CASE actingLoadStep OF
	0:
		IF NOT actingStorage.findSlot(materialID := material, atSlot => slot) THEN //load from staging table
			fail := TRUE;
			RETURN;
		END_IF
		
		IF
			actingRobot.setCommandAndWait( //perform the task
				task:= A22.LOAD_CORNER_GUARD_LOWER,
				param1:= slot,
				param2:= 0,
				param3:= 0)
		THEN
			actingLoadStep := COMPLETE;
		END_IF
		
	COMPLETE:
		loadBottomLeft := TRUE;
END_CASE
END_METHOD

METHOD PROTECTED loadBottomRight : BOOL
VAR_IN_OUT
	actingRobot : Robot;
	actingStorage : MaterialStorage;
	actingLoadStep : INT;
END_VAR
VAR_INPUT
	material : STRING;
END_VAR
VAR_OUTPUT
	fail : BOOL;
END_VAR
VAR
	slot : INT;
END_VAR
IF material = '' THEN
	loadBottomRight := TRUE;
	RETURN;
END_IF

CASE actingLoadStep OF
	0:
		IF NOT actingStorage.findSlot(materialID := material, atSlot => slot) THEN //load from staging table
			fail := TRUE;
			RETURN;
		END_IF
		
		IF
			actingRobot.setCommandAndWait( //perform the task
				task:= A22.LOAD_CORNER_GUARD_LOWER,
				param1:= slot,
				param2:= 0,
				param3:= 0)
		THEN
			actingLoadStep := COMPLETE;
		END_IF
		
	COMPLETE:
		loadBottomRight := TRUE;
END_CASE
END_METHOD

METHOD PROTECTED loadCornerCardboards : BOOL
VAR_INPUT
	pair : REFERENCE TO PositionMaterials;
END_VAR
IF cornerSetLeft = 0 THEN //LEFT SIDE
	cornerSetLeft := Surface.TOP_RIGHT;
END_IF

IF
	leftRobotCornersSequence(
		actingRobot:= robotLeft, 
		skid:= skidLeft, 
		surfaceID:= cornerSetLeft,
		loadStep:= loadStepLeft, 
		materialID:= pair.topRight, 
		foldPos0:= currentBundle.cardboardFolds[cornerSetLeft][iPair],
		foldPos1:= 0,
		fail=> )
THEN
	CASE cornerSetLeft OF
		Surface.TOP_RIGHT: 
			cornerSetLeft := Surface.TOP_LEFT;
			loadStepLeft := 0;
			
		Surface.TOP_LEFT: 
			cornerSetLeft := Surface.BOTTOM_RIGHT;
			loadStepLeft := 0;
			
		Surface.BOTTOM_RIGHT: 
			cornerSetLeft := Surface.BOTTOM_LEFT;
			loadStepLeft := 0;
			
		Surface.BOTTOM_LEFT: 
			cornerSetLeft := COMPLETE;
			loadStepLeft := COMPLETE;
			
		COMPLETE:
			//
			
	END_CASE
END_IF



IF cornerSetRight = 0 THEN //RIGHT SIDE
	cornerSetRight := Surface.TOP_RIGHT;
END_IF

IF
	rightRobotCornersSequence(
		actingRobot:= robotRight, 
		skid:= skidRight, 
		loadStep:= loadStepRight, 
		materialID:= pair.topRight, 
		surfaceID:= cornerSetRight,
		foldPos1:= currentBundle.cardboardFolds[cornerSetRight][iPair], 
		foldPos2:= 0, 
		fail=> )
THEN
	CASE cornerSetRight OF
		Surface.TOP_RIGHT: 
			cornerSetRight := Surface.BOTTOM_RIGHT;
			loadStepRight := 0;
			
		Surface.BOTTOM_RIGHT: 
			cornerSetRight := COMPLETE;			
			loadStepRight := COMPLETE;
			
		COMPLETE:
			//
			
	END_CASE
END_IF


IF cornerSetLeft = COMPLETE AND cornerSetRight = COMPLETE THEN
	loadCornerCardboards := TRUE;
	
	loadStepLeft := loadStepRight := 0;
	cornerSetLeft := cornerSetRight := 0;
END_IF
END_METHOD

METHOD PROTECTED loadCornerGuards : BOOL
VAR_INPUT
	pair : REFERENCE TO PositionMaterials;
END_VAR
VAR_OUTPUT
	fail : BOOL;
END_VAR
VAR
	leftFail : BOOL;
	rightFail : BOOL;
END_VAR
CASE loadSet OF
	0: //upper corners
		IF 
			loadCornerGuardSequence(
				actingRobot:= robotLeft, 
				robotOutputs:= robotLeftOutputs, 
				actingStorage:= skidLeft, 
				actingLoadStep:= loadStepLeft, 
				surfaceID:= Surface.TOP_LEFT, 
				material:= pair.topLeft, 
				fail=> leftFail)
			AND
			loadCornerGuardSequence(
				actingRobot:= robotRight, 
				robotOutputs:= robotRightOutputs, 
				actingStorage:= skidRight,
				actingLoadStep:= loadStepRight, 
				surfaceID:= Surface.TOP_RIGHT, 
				material:= pair.topRight, 
				fail=> rightFail)
		THEN
			loadStepLeft := loadStepRight := 0;
			loadSet := 10;
		END_IF
		
	10: //lower corners
		IF 
			loadCornerGuardSequence(
				actingRobot:= robotLeft, 
				robotOutputs:= robotLeftOutputs, 
				actingStorage:= skidLeft, 
				actingLoadStep:= loadStepLeft, 
				surfaceID:= Surface.BOTTOM_LEFT, 
				material:= pair.bottomLeft, 
				fail=> leftFail)
			AND
			loadCornerGuardSequence(
				actingRobot:= robotRight, 
				robotOutputs:= robotRightOutputs, 
				actingStorage:= skidRight,
				actingLoadStep:= loadStepRight, 
				surfaceID:= Surface.BOTTOM_RIGHT, 
				material:= pair.bottomRight, 
				fail=> rightFail)
		THEN
			loadStepLeft := loadStepRight := 0;
			loadSet := COMPLETE;
		END_IF
	
	COMPLETE:
		loadStepLeft := loadStepRight := 0;
		loadSet := 0;
		
		loadCornerGuards := TRUE;
END_CASE

fail := MAX(leftFail, rightFail);
END_METHOD

METHOD loadCornerGuardSequence : BOOL
VAR_IN_OUT
	actingRobot : Robot;
	robotOutputs : ARRAY[1..50] OF INT;
	actingStorage : MaterialStorage;
	actingLoadStep : INT;
END_VAR
VAR_INPUT
	surfaceID : Surface;
	material : STRING;
END_VAR
VAR_OUTPUT
	fail : BOOL;
END_VAR
VAR
	slot : INT;
END_VAR
IF material = '' THEN
	loadCornerGuardSequence := TRUE;
	RETURN;
END_IF

CASE actingLoadStep OF
	0:
		IF NOT actingStorage.findSlot(materialID := material, atSlot => slot) THEN //load from staging table
			fail := TRUE;
			RETURN;
		END_IF
		
		MEMSET(ADR(robotOutputs), 0, SIZEOF(robotOutputs));
		CASE surfaceID OF
			Surface.TOP_LEFT, Surface.TOP_RIGHT: 		robotOutputs[1] := A22.LOAD_CORNER_GUARD_UPPER;
			Surface.BOTTOM_LEFT, Surface.BOTTOM_RIGHT:	robotOutputs[1] := A22.LOAD_CORNER_GUARD_LOWER;
		END_CASE
		robotOutputs[2] := slot;
		
		IF actingRobot.setParamsAndWait(robotOutputs) THEN
			actingLoadStep := COMPLETE;
		END_IF
		
	COMPLETE:
		//outerSuctions[surfaceID].enable := TRUE;
		loadCornerGuardSequence := TRUE;
END_CASE
END_METHOD

METHOD PROTECTED loadFlats : BOOL
VAR_INPUT
	pair : REFERENCE TO PositionMaterials;
END_VAR
CASE loadSet OF
	0: //top and bottom
		IF 
			loadTop(robotLeft, skidLeft, loadStepLeft, pair.top, fail=> ) AND
			loadBottom(robotRight, skidRight, loadStepRight, pair.bottom, fail=> )
		THEN
			loadStepLeft := loadStepRight := 0;
			loadSet := 10;
		END_IF
		
	10: //sides
		IF 
			loadSides(robotLeft, skidLeft, loadStepLeft, pair.top, fail=> ) AND
			loadSides(robotRight, skidRight, loadStepRight, pair.bottom, fail=> )
		THEN
			loadStepLeft := loadStepRight := 0;
			loadSet := COMPLETE;
		END_IF
	
	COMPLETE:
		loadStepLeft := loadStepRight := 0;
		loadSet := 0;
		
		loadFlats := TRUE;
END_CASE
END_METHOD

METHOD loadFlatSequence : BOOL
VAR_IN_OUT
	actingRobot : Robot;
	robotOutputs : ARRAY[1..50] OF INT;
	actingStorage : MaterialStorage;
	actingLoadStep : INT;
END_VAR
VAR_INPUT
	surfaceID : Surface;
	material : STRING;
END_VAR
VAR_OUTPUT
	fail : BOOL;
END_VAR
VAR
	slot : INT;
END_VAR
IF material = '' THEN
	loadFlatSequence := TRUE;
	RETURN;
END_IF

CASE actingLoadStep OF
	0:
		IF NOT actingStorage.findSlot(materialID := material, atSlot => slot) THEN
			fail := TRUE;
			RETURN;
		END_IF
		
		MEMSET(ADR(robotOutputs), 0, SIZEOF(robotOutputs));
		CASE surfaceID OF
			Surface.TOP: 					robotOutputs[1] := A22.LOAD_CARDBOARD_TOP;
			Surface.LEFT, Surface.RIGHT: 	robotOutputs[1] := A22.LOAD_CARDBOARD_SIDE;
			Surface.BOTTOM: 				robotOutputs[1] := A22.LOAD_CARDBOARD_BOTTOM;
		END_CASE
		robotOutputs[2] := slot;
		
		IF actingRobot.setParamsAndWait(robotOutputs) THEN
			actingLoadStep := COMPLETE;
		END_IF
		
	COMPLETE:
		loadFlatSequence := TRUE;
	
END_CASE
END_METHOD

METHOD PROTECTED loadSides : BOOL
VAR_IN_OUT
	actingRobot : Robot;
	actingStorage : MaterialStorage;
	actingLoadStep : INT;
END_VAR
VAR_INPUT
	material : STRING;
END_VAR
VAR_OUTPUT
	fail : BOOL;
END_VAR
VAR
	slot : INT;
END_VAR
IF material = '' THEN
	loadSides := TRUE;
	RETURN;
END_IF

CASE actingLoadStep OF
	0:
		IF NOT actingStorage.findSlot(materialID := material, atSlot => slot) THEN
			fail := TRUE;
			RETURN;
		END_IF
		
		IF
			actingRobot.setCommandAndWait( //perform the task
				task:= A22.LOAD_CARDBOARD_SIDE,
				param1:= slot,
				param2:= 0,
				param3:= 0)
		THEN
			actingLoadStep := COMPLETE;
		END_IF
		
	COMPLETE:
		//turn suction on
		loadSides := TRUE;
END_CASE
END_METHOD

METHOD PROTECTED loadTop : BOOL
VAR_IN_OUT
	actingRobot : Robot;
	actingStorage : MaterialStorage;
	actingLoadStep : INT;
END_VAR
VAR_INPUT
	material : STRING;
END_VAR
VAR_OUTPUT
	fail : BOOL;
END_VAR
VAR
	slot : INT;
END_VAR
IF material = '' THEN
	loadTop := TRUE;
	RETURN;
END_IF

CASE actingLoadStep OF
	0:
		IF NOT actingStorage.findSlot(materialID := material, atSlot => slot) THEN //load from staging table
			fail := TRUE;
			RETURN;
		END_IF
		
		IF
			actingRobot.setCommandAndWait( //perform the task
				task:= A22.LOAD_CARDBOARD_TOP,
				param1:= slot,
				param2:= 0,
				param3:= 0)
		THEN
			actingLoadStep := COMPLETE;
		END_IF
		
	COMPLETE:
		loadTop := TRUE;
END_CASE
END_METHOD

METHOD PROTECTED loadTopLeft : BOOL
VAR_IN_OUT
	actingRobot : Robot;
	actingStorage : MaterialStorage;
	actingLoadStep : INT;
END_VAR
VAR_INPUT
	material : STRING;
END_VAR
VAR_OUTPUT
	fail : BOOL;
END_VAR
VAR
	slot : INT;
END_VAR
IF material = '' THEN
	loadTopLeft := TRUE;
	RETURN;
END_IF

CASE actingLoadStep OF
	0:
		IF NOT actingStorage.findSlot(materialID := material, atSlot => slot) THEN //load from staging table
			fail := TRUE;
			RETURN;
		END_IF
		
		IF
			actingRobot.setCommandAndWait( //perform the task
				task:= A22.LOAD_CORNER_GUARD_UPPER,
				param1:= slot,
				param2:= 0,
				param3:= 0)
		THEN
			actingLoadStep := COMPLETE;
		END_IF
		
	COMPLETE:
		loadTopLeft := TRUE;
END_CASE
END_METHOD

METHOD PROTECTED loadTopRight : BOOL
VAR_IN_OUT
	actingRobot : Robot;
	actingStorage : MaterialStorage;
	actingLoadStep : INT;
END_VAR
VAR_INPUT
	material : STRING;
END_VAR
VAR_OUTPUT
	fail : BOOL;
END_VAR
VAR
	slot : INT;
END_VAR
IF material = '' THEN
	loadTopRight := TRUE;
	RETURN;
END_IF

CASE actingLoadStep OF
	0:
		IF NOT actingStorage.findSlot(materialID := material, atSlot => slot) THEN //load from staging table
			fail := TRUE;
			RETURN;
		END_IF
		
		IF
			actingRobot.setCommandAndWait( //perform the task
				task:= A22.LOAD_CORNER_GUARD_UPPER,
				param1:= slot,
				param2:= 0,
				param3:= 0)
		THEN
			actingLoadStep := COMPLETE;
		END_IF
		
	COMPLETE:
		loadTopRight := TRUE;
END_CASE
END_METHOD

METHOD placeFrontCover : BOOL
VAR_INPUT
END_VAR
END_METHOD

METHOD PROTECTED process : BOOL
VAR
	masterLength : REAL;
	targetPos : REAL;
	targetStep : INT;
END_VAR
VAR
	maxHeight : REAL := 1000; //1000mm, 100cm, 1m tall at home pos
END_VAR
(*
VAR_INST
	resumePosition : REAL;
END_VAR
VAR CONSTANT
	wrapDelta : REAL := 5;
END_VAR
*)
//TODO: write instructions for wrapping front and back covers

IF NOT frontCoverPlaced THEN
	targetPos := 0;
	
ELSIF iPair < GVL.maxPairs THEN
	targetPos := currentPair.position;
	
ELSIF NOT backCoverPlaced AND iPair >= GVL.maxPairs THEN
	targetPos := currentBundle.length;
	
ELSIF iPair >= GVL.maxPairs THEN
	process := TRUE;
	RETURN;
	
END_IF

CASE step OF
	PLACE_FRONT_COVER:
		IF placeFrontCover() THEN
			step := RUN_TO_POSITION;
		END_IF
	
	RUN_TO_POSITION:
		IF //only load corners, flats will be PUSHed when bundle arrives at position
			directionCheckAndSet(pushConveyorPos, currentPair.position) AND 
			load(pair:= currentPair)
		THEN
			step := 10;
		END_IF
		
	LOAD_FLATS:
		IF loadFlats(pair:= currentPair) THEN
			step := PUSH;
		END_IF
		
	PUSH:
		setConveyorMode(ConveyorMode.STOP);
		(*
		IF
			NOT insertionLeft.align(targetPos:= maxHeight - currentBundle.height) OR
			NOT insertionRight.align(targetPos:= maxHeight - currentBundle.height)
		THEN
			RETURN;
		END_IF
		
		insertionLeft.press();
		insertionRight.press();
		*)
		
		IF NOT insertionLeft.contact THEN
			//insertionRight.slideOut();
			insertionLeft.traverse(direction:= MC_Negative_Direction);
			insertionLeft.press();
		END_IF
		
		IF NOT insertionRight.contact THEN
			//insertionRight.slideOut();
			insertionRight.traverse(direction:= MC_Negative_Direction);
			insertionRight.press();
		END_IF
		
		(*
		IF NOT insertionBottom.contact THEN
			insertionBottom.traverse(direction := FALSE);
		END_IF
		*)
		
		IF insertionLeft.contact AND insertionRight.contact (*AND insertionBottom.contact*) THEN		
			step := RUN_TO_WRAP_POSITION;
		END_IF
		
	RUN_TO_WRAP_POSITION:
		masterLength := GetPositionMasterLength(currentPair);
		IF iWrap >= currentPair.wrapPoints THEN
			step := COMPLETE;
			RETURN;
		END_IF
		
		IF //compare current position with wrap position
			directionCheckAndSet(
				wrapConveyorPos,
				(currentPair.position - masterLength/2) + (masterLength/(currentPair.wrapPoints + 1) * (iWrap + 1)))
		THEN
			step := WRAP_AND_RELEASE;
		END_IF
		
	WRAP_AND_RELEASE: //wrap
		setConveyorMode(ConveyorMode.STOP);
		IF wrapper.ready OR (NOT wrapper.busy AND NOT wrapper.error) THEN
			wrapper.wrap(currentPair.wrapRotations);
		END_IF
		
		IF NOT insertionLeft.home THEN
			insertionLeft.align(0);
			insertionLeft.release();
		END_IF
		
		IF NOT insertionRight.home THEN
			insertionRight.align(0);
			insertionRight.release();
		END_IF
		
		IF wrapper.done AND insertionLeft.home AND insertionRight.home (*AND insertionBottom.home*) THEN
			step := WRAP_AND_RELEASE;
		END_IF
		
	COMPLETE: //reset
		setConveyorMode(ConveyorMode.FORWARD);
		
		iPair := iPair + 1;
		IF iPair >= GVL.maxPairs THEN
			iPair := 0;
			process := TRUE;
		END_IF
		iWrap := 0;
		
		step := 0;
END_CASE
END_METHOD

METHOD PROTECTED rightRobotCornersSequence : BOOL
VAR_IN_OUT
	actingRobot : Robot;
	skid : MaterialStorage;
	loadStep : INT;
END_VAR
VAR_INPUT
	surfaceID : Surface;
	materialID : STRING;
	foldPos1 : INT;
	foldPos2 : INT;
END_VAR
VAR_OUTPUT
	fail : BOOL;
END_VAR
VAR
	slot : INT;
	
	task : INT;
	param0, param1, param2 : INT;
END_VAR
IF materialID = '' THEN
	rightRobotCornersSequence := TRUE;
	RETURN;
END_IF

CASE loadStep OF
	0: //overhead to insertion
		IF overhead = '' THEN
			RETURN;
		END_IF
		
		CASE surfaceID OF
			Surface.TOP_RIGHT:
				task := A22.LOAD_OVERHEAD_TO_UPPER_CORNER;
				
			Surface.BOTTOM_RIGHT:
				task := A22.LOAD_OVERHEAD_TO_LOWER_CORNER;
				
		END_CASE
		
		IF
			actingRobot.setCommandAndWait(
				task:= task, 
				param1:= slot, 
				param2:= foldPos1, 
				param3:= foldPos2)
		THEN
			loadStep := COMPLETE;
		END_IF
	
	COMPLETE:
		//turn on suction
		rightRobotCornersSequence := TRUE;
	
END_CASE
END_METHOD

METHOD PROTECTED robotsFailed : BOOL
VAR_INPUT
END_VAR
IF NOT robotLeft.operational OR NOT robotLeft.operational THEN
	error := TRUE;
	currentBypass := TRUE;
	robotsFailed := TRUE;
END_IF
END_METHOD

METHOD PROTECTED setOrder : BOOL
VAR_IN_OUT
	innerArray : ARRAY[*] OF PositionMaterials;
	outerArray : ARRAY[*] OF PositionMaterials;
	
	combined : ARRAY[*] OF PositionMaterials;
	
	i_inner : INT;
	i_outer : INT;
	i_combined : INT;
END_VAR
VAR
	topLength : REAL;
	leftLength : REAL;
	rightLength : REAL;
	bottomLength : REAL;
	
	topLeftLength : REAL;
	topRightLength : REAL;
	bottomLeftLength : REAL;
	bottomRightLength : REAL;
	
	outerMaterialLength : REAL;
	innerMaterialLength : REAL;
END_VAR
//if inner material is in front of outer material, inner material goes first
IF innerArray[i_inner].position <= outerArray[i_outer].position THEN

	combined[i_combined] := innerArray[i_inner];
	i_inner := i_inner + 1; //check next cardboard during next iteration
	
	setOrder := TRUE;
	RETURN;
END_IF
	
outerMaterialLength := GetPositionMasterLength(outerArray[i_outer]);
innerMaterialLength := GetPositionMasterLength(innerArray[i_inner]);

//if current inner material is too close to current outer material, place inner material first
//compare inner materials' front with outer material's back
IF (innerArray[i_inner].position - innerMaterialLength/2) < (outerArray[i_outer].position + outerMaterialLength/2) THEN
	combined[i_combined] := innerArray[i_inner];
	i_inner := i_inner + 1;
ELSE //otherwise, outer material can go
	combined[i_combined] := outerArray[i_outer];
	i_outer := i_outer + 1;
END_IF

setOrder := TRUE;
END_METHOD

METHOD PROTECTED usesProcess : BOOL
VAR
	i : INT;
END_VAR
IF materialsArr = 0 THEN
	RETURN;
END_IF

FOR i:=0 TO GVL.maxPairs BY 1 DO
	IF PositionIsValid(materialsArr[i]) THEN
		usesProcess := TRUE;
		RETURN;		
	END_IF
END_FOR
END_METHOD

END_FUNCTION_BLOCK

// ---- Sections/Concrete/ChipboardEx.TcPOU
FUNCTION_BLOCK ChipboardEx EXTENDS SectionEx
VAR
	robotLeft, robotRight : REFERENCE TO Robot;
	
	skidLeft, skidRight : REFERENCE TO MaterialStorage;
	
	toolStorageLeft, toolStorageRight : REFERENCE TO A21ToolStorage;
END_VAR
VAR
	pushSmallConveyorPos : REAL;
	pushLargeConveyorPos : REAL;
	
	topCIP : STRING;
	bottomCIP : STRING;
	
	materialsArr : POINTER TO PositionMaterials; //array of PositionMaterials
	//currentPair : REFERENCE TO PositionMaterials;	
	
	step : (RUN_TO_POSITION, LOAD_MATERIAL, PUSH, RESET);
	
	robotLeftOutputs, robotRightOutputs : ARRAY[1..50] OF INT;
END_VAR

entryRefPos := pushSmallConveyorPos;
exitRefPos := pushLargeConveyorPos;

SUPER^();

CASE status OF
	SectionStatus.IDLE:
		//RETURN;
	
	SectionStatus.ALIGNING:
		//
		
	SectionStatus.ACTIVE:
		//
		
	SectionStatus.CLEARING:
		//
		
	SectionStatus.COMPLETE:	
		//
		
	-100:
		RETURN;
		
END_CASE
	
materialsArr := ADR(currentBundle.chipboard);

loaded := 
	topCIP = materialsArr[iPair].top AND
	bottomCIP = materialsArr[iPair].bottom;
	
IF NOT(robotLeft.operational AND robotRight.operational) THEN
	currentBypass := TRUE;
END_IF

METHOD changeRobotsEOAT : BOOL
VAR_INPUT
END_VAR
IF robotLeft.tool <> sectionID THEN
	MEMSET(ADR(robotLeftOutputs), 0, SIZEOF(robotLeftOutputs));
	robotLeftOutputs[1] := A21.TOOL_CHANGE_CHIPBOARD;
	robotLeft.setParamsAndWait(robotLeftOutputs);
END_IF

IF robotRight.tool <> sectionID THEN
	MEMSET(ADR(robotRightOutputs), 0, SIZEOF(robotRightOutputs));
	robotRightOutputs[1] := A21.TOOL_CHANGE_CHIPBOARD;
	robotRight.setParamsAndWait(robotRightOutputs);
END_IF

changeRobotsEOAT := robotLeft.tool = sectionID AND robotRight.tool = sectionID;
END_METHOD

METHOD initHardware : BOOL
conveyors := ADR(allConveyors);

robotLeft REF= robots[1];
robotRight REF= robots[2];

skidLeft REF= chipboardSkidLeft;
skidRight REF= chipboardSkidRight;
END_METHOD

METHOD PROTECTED load : BOOL
VAR_INPUT
	pair : REFERENCE TO PositionMaterials;
END_VAR
(*
top:
	grab chipboard
	move chipboard to top

bottom:
	grab chipboard and lower conveyor
	move chipboard to lowered conveyor
	which conveyor depends on size of chipboard
	raise conveyor
*)
IF NOT (robotLeft.reserve(sectionID) AND robotRight.reserve(sectionID)) THEN
	RETURN;
END_IF

IF NOT (robotLeft.tool = sectionID AND robotRight.tool = sectionID) THEN //robots have wrong tool
	changeRobotsEOAT(); //wait for robots to finish changing tools
	RETURN;
END_IF
//continues once both robots have correct tool

CASE loadSet OF
	0: //top and bottom
		IF 
			loadingSequence(
				actingRobot:= robotLeft, 
				robotOutputs:= robotLeftOutputs, 
				storage:= skidLeft, 
				loadStep:= loadStepLeft, 
				surfaceID:= Surface.TOP,
				material:= pair.top, 
				fail=> )
			AND
			loadingSequence(
				actingRobot:= robotRight, 
				robotOutputs:= robotRightOutputs, 
				storage:= skidRight, 
				loadStep:= loadStepRight, 
				surfaceID:= Surface.TOP,
				material:= pair.bottom, 
				fail=> )
		THEN
			loadStepLeft := loadStepRight := 0;
			loadSet := 10;
		END_IF
		
	10 : //recovery
		IF robotLeft.operational AND NOT robotRight.operational THEN //left ok, right fail
			IF
				loadingSequence(
					actingRobot:= robotLeft, 
					robotOutputs:= robotLeftOutputs, 
					storage:= skidLeft, 
					loadStep:= loadStepLeft, 
					surfaceID:= Surface.BOTTOM,
					material:= pair.top, 
					fail=> ) //load bottom with left robot
			THEN
				step := COMPLETE;
			END_IF
			
		ELSIF NOT robotLeft.operational AND robotRight.operational THEN //left fail, right ok
			IF
				loadingSequence(
					actingRobot:= robotRight, 
					robotOutputs:= robotRightOutputs, 
					storage:= skidRight, 
					loadStep:= loadStepRight, 
					surfaceID:= Surface.TOP,
					material:= pair.bottom, 
					fail=> ) //load top with right robot
			THEN
				step := COMPLETE;
			END_IF
			
		ELSE
			error := TRUE;
			currentBypass := TRUE;
				
		END_IF
		
		loadSet := COMPLETE;
		
	COMPLETE:
		loadSet := 0;
		
		loaded := 
			topCip = pair.top AND
			bottomCip = pair.bottom;
			
		robotLeft.release(sectionID);
		robotRight.release(sectionID);
			
		load := TRUE;
END_CASE
END_METHOD

METHOD loadBottom : BOOL
VAR_IN_OUT
	actingRobot : Robot;
	robotReserved : BOOL;
	robotOutputs : ARRAY[1..50] OF INT;
	actingStorage : MaterialStorage;
	actingLoadStep : INT;
END_VAR
VAR_INPUT
	material : STRING;
END_VAR
VAR_OUTPUT
	fail : BOOL;
END_VAR
VAR
	done : BOOL;
END_VAR
VAR
	slot : INT;
END_VAR
IF material = '' THEN
	step := COMPLETE;
END_IF

IF actingLoadStep <> COMPLETE AND_THEN NOT actingRobot.reserve(sectionID) THEN
	RETURN;
END_IF

CASE actingLoadStep OF
	0:
		IF NOT actingStorage.findSlot(materialID := material, atSlot => slot) THEN
			fail := TRUE;
			RETURN;
		END_IF
		
		MEMSET(ADR(robotOutputs), 0, SIZEOF(robotOutputs));
		robotOutputs[1] := A21.GET_CHIPBOARD_FROM_SKID;
		robotOutputs[2] := slot;
		
		IF actingRobot.setParamsAndWait(robotOutputs) THEN
			actingLoadStep := 10;
		END_IF
		
	10:
		MEMSET(ADR(robotOutputs), 0, SIZEOF(robotOutputs));
		robotOutputs[1] := A21.PLACE_CHIPBOARD_TO_BOTTOM;
		robotOutputs[2] := slot;
		
		IF actingRobot.setParamsAndWait(robotOutputs) THEN
			actingLoadStep := 10;
		END_IF
		
	COMPLETE:
		actingRobot.release(sectionID);
		loadBottom := TRUE;
		
END_CASE
END_METHOD

METHOD loadingSequence : BOOL
VAR_IN_OUT
	actingRobot : Robot;
	robotOutputs : ARRAY[1..50] OF INT;
	storage : MaterialStorage;
	loadStep : INT;
END_VAR
VAR_INPUT
	surfaceID : Surface;
	material : STRING;
END_VAR
VAR_OUTPUT
	fail : BOOL;
END_VAR
VAR
	slot : INT;
END_VAR
IF material = '' THEN
	loadingSequence := TRUE;
	RETURN;
END_IF

CASE loadStep OF
	0:
		IF NOT storage.findSlot(materialID := material, atSlot => slot) THEN
			fail := TRUE;
			RETURN;
		END_IF
		
		MEMSET(ADR(robotOutputs), 0, SIZEOF(robotOutputs));
		robotOutputs[1] := A21.GET_CHIPBOARD_FROM_SKID;
		robotOutputs[2] := slot;
		
		CASE surfaceID OF
			Surface.TOP:
				IF actingRobot.setParamsAndWait(robotOutputs) THEN
					loadStep := 10;
				END_IF
				
			Surface.BOTTOM:
				//lower conveyor
				IF actingRobot.setParamsAndWait(robotOutputs) (*AND conveyor lowered*) THEN
					loadStep := 10;
				END_IF
			
		END_CASE
		
	10:
		MEMSET(ADR(robotOutputs), 0, SIZEOF(robotOutputs));
		CASE surfaceID OF
			Surface.TOP: 					robotOutputs[1] := A21.PLACE_CHIPBOARD_TO_TOP;
			Surface.BOTTOM: 				robotOutputs[1] := A21.PLACE_CHIPBOARD_TO_BOTTOM;
		END_CASE
		robotOutputs[2] := slot;
		
		IF actingRobot.setParamsAndWait(robotOutputs) THEN
			loadStep := 10;
		END_IF
		
	COMPLETE:
		actingRobot.release(sectionID);
		loadingSequence := TRUE;
		
END_CASE
END_METHOD

METHOD loadTop : BOOL
VAR_IN_OUT
	actingRobot : Robot;
	robotOutputs : ARRAY[1..50] OF INT;
	actingStorage : MaterialStorage;
	actingLoadStep : INT;
END_VAR
VAR_INPUT
	material : STRING;
END_VAR
VAR_OUTPUT
	fail : BOOL;
END_VAR
VAR
	slot : INT;
END_VAR
IF actingLoadStep <> COMPLETE AND_THEN NOT actingRobot.reserve(sectionID) THEN
	RETURN;
END_IF

CASE actingLoadStep OF
	0: //grab chipboard
		IF NOT actingStorage.findSlot(materialID := material, atSlot => slot) THEN
			fail := TRUE;
			RETURN;
		END_IF
		
		MEMSET(ADR(robotOutputs), 0, SIZEOF(robotOutputs));
		robotOutputs[1] := A21.GET_CHIPBOARD_FROM_SKID;
		robotOutputs[2] := slot;
		
		IF actingRobot.setParamsAndWait(robotOutputs) THEN
			actingLoadStep := 10;
		END_IF
		
	10: //load chipboard
		MEMSET(ADR(robotOutputs), 0, SIZEOF(robotOutputs));
		robotOutputs[1] := A21.PLACE_CHIPBOARD_TO_TOP;
		robotOutputs[2] := slot;
		
		IF actingRobot.setParamsAndWait(robotOutputs) THEN
			actingLoadStep := 10;
		END_IF
		
	COMPLETE:
		actingRobot.release(sectionID);
		loadTop := TRUE;
		
END_CASE
END_METHOD

METHOD PROTECTED process : BOOL
VAR
	currentPair : REFERENCE TO PositionMaterials REF= materialsArr[iPair];
END_VAR
VAR_INST
	cmdSent : BOOL;
	
	test : BOOL;
	
	i : INT;
	conveyorsExtended : BOOL := TRUE;
END_VAR
IF iPair >= GVL.maxPairs THEN
	process := TRUE;
	RETURN;
END_IF

CASE step OF
	RUN_TO_POSITION: //free run until position reached
		IF directionCheckAndSet(pushSmallConveyorPos, currentPair.position) THEN
			step := PUSH;
		END_IF
		
	LOAD_MATERIAL: //loading must be done when bundle reaches position, not before
		setConveyorMode(ConveyorMode.STOP); //request stop at position
		IF load(currentPair) THEN
			step := PUSH;
		END_IF
	
	PUSH: //push materials
		setConveyorMode(ConveyorMode.STOP); //request stop at position
		FOR i:=firstConveyor TO lastConveyor BY 1 DO
			IF NOT conveyors[i].extended THEN
				conveyors[i].extend();
			END_IF
			conveyorsExtended := MIN(conveyorsExtended, conveyors[i].extended);
		END_FOR
		
		IF conveyorsExtended THEN
			step := RESET;
		END_IF
		
	RESET: //finished at this position, reset
		setConveyorMode(ConveyorMode.FORWARD);
		cmdSent := FALSE;
		
		iPair := iPair + 1;
		
		step := 0;
END_CASE
END_METHOD

METHOD PROTECTED usesProcess : BOOL
VAR
	i : INT;
END_VAR
IF materialsArr = 0 THEN
	RETURN;
END_IF

FOR i:=0 TO GVL.maxPairs BY 1 DO
	IF PositionIsValid(materialsArr[i]) THEN
		usesProcess := TRUE;
		RETURN;		
	END_IF
END_FOR
END_METHOD

END_FUNCTION_BLOCK

// ---- Sections/Concrete/WoodBunkEx.TcPOU
FUNCTION_BLOCK WoodBunkEx EXTENDS SectionEx
VAR //references to objects imported from Hardware GVL - using references instead of VAR_EXTERNAL or direct access allows local renaming
	robotLeft, robotRight : REFERENCE TO Robot;
	
	stagingTableLeft, stagingTableRight : REFERENCE TO WoodBunkTable;
	magazineLeft, magazineRight: REFERENCE TO MaterialStorage;
	
	strapper : REFERENCE TO StrapMachine;
	
	insertionLeft, insertionRight : REFERENCE TO Insertion;
	insertionBottom : REFERENCE TO AirPiston;
	
	toolStorageLeft, toolStorageRight : REFERENCE TO A21ToolStorage;
END_VAR
VAR
	conveyorPos : REAL;
	
	insertionSlots : ARRAY[Surface.TOP..Surface.BOTTOM] OF STRING;
	
	materialsArr : POINTER TO PositionMaterials; //array of PositionMaterials
	currentPair : REFERENCE TO PositionMaterials;
	
	stagingMaterial : STRING; //ex: currentPair.left
	currentMaterial : STRING; //ex: WDS18_WDS20 --> WDS18, then WDS20
	
	stagingTemplateReady : BOOL;
	stagingTemplateLeft : WoodBunkTable;
	stagingTemplateRight : WoodBunkTable;
	
	step : (RUN_TO_POSITION, PUSH, RUN_TO_STRAP, STRAP, RELEASE, RESET);
	
	//for staging use
	stageSet : INT;	
	stageStepLeft, stageStepRight : INT;
	iStagingSlotLeft, iStagingSlotRight : INT;
	
	robotLeftOutputs, robotRightOutputs : ARRAY[1..50] OF INT;
END_VAR
VAR
	tempInspectionSuite : VisionSuite; //send/receive from TcpServer
	leftInspectionFrame, rightInspectionFrame : VisionFrame; //parsed from above
END_VAR
VAR CONSTANT
	leftCamera : INT := 1;
	rightCamera : INT := 2;
END_VAR

entryRefPos := conveyorPos;
exitRefPos := conveyorPos;

SUPER^();

CASE status OF
	SectionStatus.IDLE:
		//RETURN;
	
	SectionStatus.ALIGNING:
		//
		
	SectionStatus.ACTIVE:
		//
		
	SectionStatus.CLEARING:
		stagingTemplateReady := FALSE;
		
	SectionStatus.COMPLETE:	
		//
		
	-100:
		RETURN;
		
END_CASE

materialsArr := ADR(currentBundle.woodBunk);

loaded := 
	insertionSlots[Surface.TOP] = materialsArr[iPair].top AND
	insertionSlots[Surface.LEFT] = materialsArr[iPair].left AND
	insertionSlots[Surface.RIGHT] = materialsArr[iPair].right AND
	insertionSlots[Surface.BOTTOM] = materialsArr[iPair].bottom;
	
//bundle needs this section's materials, and either robot failed
IF usesProcess() AND NOT(robotLeft.operational AND robotRight.operational) THEN 

	currentBypass := TRUE;
	RETURN;
END_IF //otherwise, carry over bypass from prev section

stage();

METHOD changeRobotsEOAT : BOOL
VAR_INPUT
END_VAR
IF robotLeft.tool <> sectionID THEN
	MEMSET(ADR(robotLeftOutputs), 0, SIZEOF(robotLeftOutputs));
	robotLeftOutputs[1] := A21.TOOL_CHANGE_CHIPBOARD;
	robotLeft.setParamsAndWait(robotLeftOutputs);
END_IF

IF robotRight.tool <> sectionID THEN
	MEMSET(ADR(robotRightOutputs), 0, SIZEOF(robotRightOutputs));
	robotRightOutputs[1] := A21.TOOL_CHANGE_CHIPBOARD;
	robotRight.setParamsAndWait(robotRightOutputs);
END_IF

changeRobotsEOAT := robotLeft.tool = sectionID AND robotRight.tool = sectionID;
END_METHOD

METHOD PROTECTED createStagingTemplate : BOOL
VAR
	remainingMaterial : STRING;
	splitMaterial : STRING;
	
	i : INT;
END_VAR
FOR i:=0 TO GVL.maxPairs BY 1 DO //iterate through all pairs and autofill the template
	//LEFT TABLE
	remainingMaterial := materialsArr[i].top;
	WHILE FIND(remainingMaterial, '_') > 0 DO //until no underscore found
		splitCombinedMaterials(remainingMaterial, splitMaterial);
		stagingTemplateLeft.autofill(splitMaterial);
	END_WHILE
	stagingTemplateLeft.autofill(remainingMaterial);
	
	remainingMaterial := materialsArr[i].left;
	WHILE FIND(remainingMaterial, '_') > 0 DO
		splitCombinedMaterials(remainingMaterial, splitMaterial);
		stagingTemplateLeft.autofill(splitMaterial);
	END_WHILE
	stagingTemplateLeft.autofill(remainingMaterial);
	
	//RIGHT TABLE
	remainingMaterial := materialsArr[i].right;
	WHILE FIND(remainingMaterial, '_') > 0 DO
		splitCombinedMaterials(remainingMaterial, splitMaterial);
		stagingTemplateRight.autofill(splitMaterial);
	END_WHILE
	stagingTemplateRight.autofill(remainingMaterial);
	
	remainingMaterial := materialsArr[i].bottom;
	WHILE FIND(remainingMaterial, '_') > 0 DO
		splitCombinedMaterials(remainingMaterial, splitMaterial);
		stagingTemplateRight.autofill(splitMaterial);
	END_WHILE
	stagingTemplateRight.autofill(remainingMaterial);
END_FOR
END_METHOD

METHOD findOpenSlot : BOOL
VAR_INPUT
	materialCode : STRING;
END_VAR
VAR_OUTPUT
	openSlot : INT := 0;
END_VAR
(*
IF FIND(materialCode, 'WDW') > 0 THEN //top wide, load in slot 0-1
	FOR i:=1 TO 2 BY 1 DO
		IF stageTableLeft[i] = '' THEN
			findOpenSlot := TRUE;
			openSlot := i;
			RETURN;
		END_IF
	END_FOR
	
ELSIF FIND(materialCode, 'WDT') > 0 OR FIND(materialCode, 'WDS') > 0 THEN //top std and sides, load in slot 2-9
	FOR i:=3 TO 10 BY 1 DO
		IF stageTableLeft[i] = '' THEN
			findOpenSlot := TRUE;
			openSlot := i;
			RETURN;
		END_IF
	END_FOR
	
END_IF
*)
END_METHOD

METHOD initHardware : BOOL
conveyors := ADR(allConveyors);

robotLeft REF= robots[1];
robotRight REF= robots[2];

strapper REF= strapperA21;

insertionLeft REF= insertionA21Left;
insertionLeft REF= insertionA21Right;

stagingTableLeft REF= stagingTableLeft;
stagingTableRight REF= stagingTableRight;

magazineLeft REF= woodBunkMagazineLeft;
magazineRight REF= woodBunkMagazineRight;

(*
strapper REF= Hardware.strapper;

insertionLeft REF= Hardware.insertionWoodBunkSides[Surface.LEFT];
insertionLeft REF= Hardware.insertionWoodBunkSides[Surface.RIGHT];

stagingTableLeft REF= Hardware.stagingTable[Surface.LEFT];
stagingTableRight REF= Hardware.stagingTable[Surface.RIGHT];

magazineLeft REF= Hardware.woodBunkMagazine[Surface.LEFT];
magazineRight REF= Hardware.woodBunkMagazine[Surface.RIGHT];
*)
END_METHOD

METHOD PROTECTED load : BOOL
VAR_INPUT
	pair : REFERENCE TO PositionMaterials;
END_VAR
IF NOT robotLeft.operational OR NOT robotLeft.operational THEN
	error := TRUE;
	
	currentBypass := TRUE;
	RETURN;
END_IF

IF NOT (robotLeft.reserve(sectionID) AND robotRight.reserve(sectionID)) THEN
	RETURN;
END_IF

IF NOT (robotLeft.tool = sectionID AND robotRight.tool = sectionID) THEN //robots have wrong tool
	changeRobotsEOAT(); //wait for robots to finish changing tools
	RETURN;
END_IF


CASE loadSet OF
	0: //top and bottom
		IF 
			loadingSequence(
				actingRobot:= robotLeft, 
				robotOutputs:= robotLeftOutputs, 
				stagingTable:= stagingTableLeft, 
				loadStep:= loadStepLeft, 
				surfaceID:= Surface.TOP, 
				material:= pair.top, 
				fail=> )
			AND
			loadingSequence(
				actingRobot:= robotRight, 
				robotOutputs:= robotRightOutputs, 
				stagingTable:= stagingTableRight, 
				loadStep:= loadStepRight, 
				surfaceID:= Surface.BOTTOM, 
				material:= pair.bottom, 
				fail=> )
		THEN
			loadStepLeft := loadStepRight := 0;
			loadSet := 10;
		END_IF
		
	10: //sides
		IF
			loadingSequence(
				actingRobot:= robotLeft, 
				robotOutputs:= robotLeftOutputs, 
				stagingTable:= stagingTableLeft, 
				loadStep:= loadStepLeft, 
				surfaceID:= Surface.LEFT, 
				material:= pair.left, 
				fail=> )
			AND
			loadingSequence(
				actingRobot:= robotRight, 
				robotOutputs:= robotRightOutputs, 
				stagingTable:= stagingTableRight, 
				loadStep:= loadStepRight, 
				surfaceID:= Surface.RIGHT, 
				material:= pair.right, 
				fail=> )
		THEN
			loadStepLeft := loadStepRight := 0;
			loadSet := COMPLETE;
		END_IF
		
	COMPLETE:
		loadSet := 0;
		loadStepLeft := loadStepRight := 0;
		
		loaded := 
			insertionSlots[Surface.TOP] = materialsArr[iPair].top AND
			insertionSlots[Surface.LEFT] = materialsArr[iPair].left AND
			insertionSlots[Surface.RIGHT] = materialsArr[iPair].right AND
			insertionSlots[Surface.BOTTOM] = materialsArr[iPair].bottom;
		
		robotLeft.release(sectionID);
		robotRight.release(sectionID);
		
		load := TRUE;
END_CASE
END_METHOD

METHOD loadBottom : BOOL
VAR_IN_OUT //acting refers to which robot is performing the task, if the designated robot fails the other may take over
	actingRobot : Robot;
	robotOutputs : ARRAY[1..50] OF INT;
	actingStagingTable : WoodBunkTable;
	actingLoadStep : INT;
END_VAR
VAR_INPUT
	material : STRING;
END_VAR
VAR_OUTPUT
	fail : BOOL;
END_VAR
VAR
	slot : INT;
END_VAR
IF
	actingLoadStep <> COMPLETE AND_THEN
	NOT actingRobot.reserve(sectionID)
THEN
	RETURN;
END_IF

CASE actingLoadStep OF
	0:
		IF NOT actingStagingTable.findSlot(materialID := material, atSlot => slot) THEN
			fail := TRUE;
			RETURN;
		END_IF
		
		MEMSET(ADR(robotOutputs), 0, SIZEOF(robotOutputs));
		robotOutputs[1] := A21.LOAD_BUNK_TO_BOTTOM;
		robotOutputs[2] := slot;
		
		IF actingRobot.setParamsAndWait(robotOutputs) THEN
			actingLoadStep := COMPLETE;
		END_IF
		
	COMPLETE:
		//turn suction on
		actingRobot.release(sectionID);
		loadBottom := TRUE;
END_CASE
END_METHOD

METHOD loadingSequence : BOOL
VAR_IN_OUT
	actingRobot : Robot;
	robotOutputs : ARRAY[1..50] OF INT;
	stagingTable : WoodBunkTable;
	loadStep : INT;
END_VAR
VAR_INPUT
	surfaceID : Surface;
	material : STRING;
END_VAR
VAR_OUTPUT
	fail : BOOL;
END_VAR
VAR
	slot : INT;
END_VAR
IF material = '' THEN
	loadingSequence := TRUE;
	RETURN;
END_IF

CASE loadStep OF
	0:
		IF NOT stagingTable.findSlot(materialID := material, atSlot => slot) THEN
			fail := TRUE;
			RETURN;
		END_IF
		
		MEMSET(ADR(robotOutputs), 0, SIZEOF(robotOutputs));
		CASE surfaceID OF
			Surface.TOP: 					robotOutputs[1] := A21.LOAD_BUNK_TO_TOP;
			Surface.LEFT, Surface.RIGHT: 	robotOutputs[1] := A21.LOAD_BUNK_TO_SIDE;
			Surface.BOTTOM: 				robotOutputs[1] := A21.LOAD_BUNK_TO_BOTTOM;
		END_CASE
		robotOutputs[2] := slot;
		
		IF actingRobot.setParamsAndWait(robotOutputs) THEN
			loadStep := COMPLETE;
		END_IF
		
	COMPLETE:
		//turn suction on
		actingRobot.release(sectionID);
		loadingSequence := TRUE;
		
END_CASE
END_METHOD

METHOD loadSides : BOOL
VAR_IN_OUT //acting refers to which robot is performing the task, if the designated robot fails the other may take over
	actingRobot : Robot;
	robotOutputs : ARRAY[1..50] OF INT;
	actingStagingTable : WoodBunkTable;
	actingLoadStep : INT;
END_VAR
VAR_INPUT
	material : STRING;
END_VAR
VAR_OUTPUT
	fail : BOOL;
END_VAR
VAR
	slot : INT;
END_VAR
IF
	actingLoadStep <> COMPLETE AND_THEN
	NOT actingRobot.reserve(sectionID)
THEN
	RETURN;
END_IF

CASE actingLoadStep OF
	0:
		IF NOT actingStagingTable.findSlot(materialID := material, atSlot => slot) THEN
			fail := TRUE;
			RETURN;
		END_IF
		
		MEMSET(ADR(robotOutputs), 0, SIZEOF(robotOutputs));
		robotOutputs[1] := A21.LOAD_BUNK_TO_SIDE;
		robotOutputs[2] := slot;
		
		IF actingRobot.setParamsAndWait(robotOutputs) THEN
			actingLoadStep := COMPLETE;
		END_IF
		
	COMPLETE:
		//turn suction on
		actingRobot.release(sectionID);
		loadSides := TRUE;
END_CASE
END_METHOD

METHOD loadTop : BOOL
VAR_IN_OUT //acting refers to which robot is performing the task, if the designated robot fails the other may take over
	actingRobot : Robot;
	robotOutputs : ARRAY[1..50] OF INT;
	actingStagingTable : WoodBunkTable;
	actingLoadStep : INT;
END_VAR
VAR_INPUT
	material : STRING;
END_VAR
VAR_OUTPUT
	fail : BOOL;
END_VAR
VAR
	slot : INT;
END_VAR
IF
	actingLoadStep <> COMPLETE AND_THEN
	NOT actingRobot.reserve(sectionID)
THEN
	RETURN;
END_IF

CASE actingLoadStep OF
	0:
		IF NOT actingStagingTable.findSlot(materialID := material, atSlot => slot) THEN
			fail := TRUE;
			RETURN;
		END_IF
		
		MEMSET(ADR(robotOutputs), 0, SIZEOF(robotOutputs));
		robotOutputs[1] := A21.LOAD_BUNK_TO_TOP;
		robotOutputs[2] := slot;
		
		IF actingRobot.setParamsAndWait(robotOutputs) THEN
			actingLoadStep := COMPLETE;
		END_IF
		
	COMPLETE:
		//turn suction on
		actingRobot.release(sectionID);
		loadTop := TRUE;
END_CASE
END_METHOD

METHOD PROTECTED process : BOOL
VAR
	currentPair : REFERENCE TO PositionMaterials REF= materialsArr[iPair];
END_VAR
IF iPair >= GVL.maxPairs THEN
	process := TRUE;
	RETURN;
END_IF

IF NOT PositionIsValid(pair:= currentPair) THEN
	step := 0;
	iPair := iPair + 1;
	RETURN;
END_IF

CASE step OF
	RUN_TO_POSITION: //free run until position reached
		IF directionCheckAndSet(conveyorPos, currentPair.position) AND load(pair:= currentPair) THEN
			step := PUSH;
		END_IF

	PUSH: //push command
		setConveyorMode(ConveyorMode.STOP);
		IF
			NOT insertionLeft.align(currentBundle.height/2) OR
			NOT insertionRight.align(currentBundle.height/2)
		THEN
			RETURN;
		END_IF
		
		insertionLeft.press();
		insertionRight.press();
		insertionBottom.slideIn();
		
		IF insertionLeft.contact AND insertionRight.contact AND insertionBottom.contact THEN		
			step := STRAP;
		END_IF
		
	STRAP: //strap command
		setConveyorMode(ConveyorMode.STOP);
		IF strapper.ready OR (NOT strapper.busy AND NOT strapper.error) THEN
			strapper.strap();
		END_IF
		
		IF strapper.done THEN
			step := RELEASE;
		END_IF
		
	RELEASE: //release command
		setConveyorMode(ConveyorMode.STOP);
		
		IF NOT insertionLeft.home THEN
			insertionLeft.align(0);
			insertionLeft.release();
		END_IF
		
		IF NOT insertionRight.home THEN
			insertionRight.align(0);
			insertionRight.release();
		END_IF
		
		IF insertionLeft.home AND insertionRight.home THEN
			step := RESET;
		END_IF
		
	RESET: //reset
		setConveyorMode(ConveyorMode.FORWARD);
		iPair := iPair + 1;
		
		step := 0;
		
END_CASE
END_METHOD

METHOD splitCombinedMaterials : BOOL
VAR_IN_OUT
	materialID : STRING;
	splitMaterial : STRING;
END_VAR
VAR
	i : INT;
END_VAR
FindAndSplitChar(
	sSeparatorChar:= '_', 
	pSrcString:= ADR(materialID), 
	pLeftString:= ADR(splitMaterial), 
	nLeftSize:= SIZEOF(splitMaterial), 
	pRightString:= ADR(materialID), 
	nRightSize:= SIZEOF(materialID), 
	bSearchFromRight:= FALSE);
END_METHOD

METHOD stage : BOOL
//robot reservation needs to be constantly checked so it is not in the state machine
IF NOT (robotLeft.reserve(sectionID) AND robotRight.reserve(sectionID)) THEN
	RETURN;
END_IF

IF NOT (robotLeft.tool = sectionID AND robotRight.tool = sectionID) THEN //robots have wrong tool
	changeRobotsEOAT(); //wait for robots to finish changing tools
	RETURN;
END_IF

CASE stageSet OF
	0: //create staging template
		createStagingTemplate();
		stageSet := 10;
	
	10: //staging sequence
		IF TcpServer1Vision.fetch(tempInspectionSuite.data) THEN
			(*
				1 - parse
				2 - determine if the camera number is for left or right staging
				3 - copy into appropriate frame
			*)
			MEMCPY(
				ADR(tempInspectionSuite.json),
				ADR(tempInspectionSuite.data),
				MIN( SIZEOF(tempInspectionSuite.json), SIZEOF(tempInspectionSuite.data) ));
			
			VisionJsonParser(
				jsonString:= tempInspectionSuite.json,
				visionData=> );
			
			IF NOT FrameIsValid(tempInspectionSuite.frame) THEN
				//
			
			ELSIF tempInspectionSuite.frame.CameraNumber = leftCamera THEN
				leftInspectionFrame := tempInspectionSuite.frame;
				
			ELSIF tempInspectionSuite.frame.CameraNumber = rightCamera THEN
				rightInspectionFrame := tempInspectionSuite.frame;
				
			END_IF
		END_IF
		

		IF
			stagingSequence(
				template:= stagingTemplateLeft, 
				magazine:= magazineLeft, 
				table:= stagingTableLeft, 
				stagingSlot:= iStagingSlotLeft,
				actingRobot:= robotLeft, 
				robotOutputs:= robotLeftOutputs,
				inspectionFrame:= leftInspectionFrame, 
				actingStep:= stageStepLeft, 
				camera:= leftCamera, 
				fail=> )
			AND
			stagingSequence(
				template:= stagingTemplateRight, 
				magazine:= magazineRight, 
				table:= stagingTableRight, 
				stagingSlot:= iStagingSlotRight,
				actingRobot:= robotRight, 
				robotOutputs:= robotRightOutputs,
				inspectionFrame:= rightInspectionFrame, 
				actingStep:= stageStepRight, 
				camera:= rightCamera, 
				fail=> )
		THEN
			stageStepLeft := stageStepRight := 0;
			iStagingSlotLeft := iStagingSlotRight := 0;
			
			stageSet := COMPLETE;
		END_IF
		
	COMPLETE:
		stageSet := 0;
		stageStepLeft := stageStepRight := 0;
		
		robotLeft.release(sectionID);
		robotRight.release(sectionID);
		
		stage := TRUE;
		
END_CASE
END_METHOD

METHOD stageLeft : BOOL
VAR_IN_OUT
	template : WoodBunkTable;
	magazine : MaterialStorage;
	table : WoodBunkTable;
	actingStagingSlot : INT;
	actingRobot : Robot;
	robotOutputs : ARRAY[1..50] OF INT;
	actingFrame : VisionFrame;
	actingStep : INT;
END_VAR
VAR_INPUT
	camera : INT;
END_VAR
VAR_OUTPUT
	fail : BOOL;
END_VAR
VAR
	finished : BOOL;
	slot : INT;
	templateArr : POINTER TO STRING;
END_VAR
VAR CONSTANT
	WIP : INT := 0;
	PASSED : INT := 1;
	FAILED : INT := 2;
END_VAR
IF table.isFull() OR actingStagingSlot > 10 THEN
	stageLeft := TRUE;
	RETURN;
END_IF

templateArr := template.getSlotsAsArray();

//follow the template as is
IF NOT magazine.findSlot(materialID:= templateArr[actingStagingSlot], atSlot => slot) THEN
	fail := TRUE;
	RETURN;
END_IF

IF actingStep > 0 THEN
	finished := actingRobot.setCommandAndWait(A21.STAGE_BUNK, slot, actingStagingSlot, 0);
END_IF

CASE actingStep OF
	0: //command
		IF actingRobot.inputs[5].10 THEN
			actingStep := 10;
		END_IF
		
	10: //request inspection
		tempInspectionSuite.frame.MaterialID := templateArr[actingStagingSlot];
		tempInspectionSuite.frame.CheckFor := 'ORIENTATION';
		tempInspectionSuite.frame.CameraNumber := camera;
	
		CreateJsonDocumentAuto(
			visionFrameData:= tempInspectionSuite.frame, 
			jsonDocument=> tempInspectionSuite.json);
		
		MEMCPY(
			ADR(tempInspectionSuite.data), 
			ADR(tempInspectionSuite.json), 
			MIN( SIZEOF(tempInspectionSuite.data), SIZEOF(tempInspectionSuite.json) ));
			
		TcpServer1Vision.queue(tempInspectionSuite.data);
		
		actingStep := 20;
	
	20: //fetch inspection data and parse
		actingRobot.setCommandAndWait(A21.STAGE_BUNK, slot, actingStagingSlot, 0);
		robotOutputs[4] := 0;
		
		IF NOT FrameIsValid(actingFrame) THEN
			RETURN;
		END_IF
		
		IF actingFrame.SuccessFlag = 1 THEN
			robotOutputs[4] := PASSED;
		ELSE
			robotOutputs[4] := FAILED;
		END_IF
		actingStep := 30;
		
	30: //finish command
		IF finished THEN
			IF actingFrame.SuccessFlag = 1 THEN
				actingStagingSlot := actingStagingSlot + 1;
			END_IF
			
			actingStep := 0;
		END_IF
END_CASE
END_METHOD

METHOD stageRight : BOOL
VAR_IN_OUT
	template : WoodBunkTable;
	magazine : MaterialStorage;
	table : WoodBunkTable;
	actingStagingSlot : INT;
	actingRobot : Robot;
	actingFrame : VisionFrame;
	actingStep : INT;
END_VAR
VAR_INPUT
	camera : INT;
END_VAR
VAR_OUTPUT
	fail : BOOL;
END_VAR
VAR
	finished : BOOL;
	robotOutputs : POINTER TO INT;
	
	slot : INT;
	templateArr : POINTER TO STRING;
	
END_VAR
IF table.isFull() OR actingStagingSlot > 10 THEN
	stageRight := TRUE;
	RETURN;
END_IF

templateArr := template.getSlotsAsArray();

//follow the template as is
IF NOT magazine.findSlot(materialID:= templateArr[actingStagingSlot], atSlot => slot) THEN
	fail := TRUE;
	RETURN;
END_IF

IF actingStep > 0 THEN
	finished := actingRobot.setCommandAndWait(A21.STAGE_BUNK, slot, actingStagingSlot, 0);
END_IF

CASE actingStep OF
	0: //command
		IF actingRobot.inputs[5].10 THEN
			actingStep := 10;
		END_IF
		
	10: //send inspection data
		tempInspectionSuite.frame.MaterialID := templateArr[actingStagingSlot];
		tempInspectionSuite.frame.CheckFor := 'ORIENTATION';
		tempInspectionSuite.frame.CameraNumber := camera;
	
		CreateJsonDocumentAuto(
			visionFrameData:= tempInspectionSuite.frame, 
			jsonDocument=> tempInspectionSuite.json);
		
		MEMCPY( //data = json
			ADR(tempInspectionSuite.data), 
			ADR(tempInspectionSuite.json), 
			MIN( SIZEOF(tempInspectionSuite.data), SIZEOF(tempInspectionSuite.json) ));
			
		TcpServer1Vision.queue(tempInspectionSuite.data);
		
		actingStep := 20;
	
	20: //fetch inspection data and parse
		actingRobot.setCommandAndWait(A21.STAGE_BUNK, slot, actingStagingSlot, 0);
		robotOutputs[11] := 0;
		
		IF NOT FrameIsValid(actingFrame) THEN
			RETURN;
		END_IF
		
		IF actingFrame.SuccessFlag = 1 THEN
			robotOutputs[11] := 1;
		ELSE
			robotOutputs[11] := 2;
		END_IF
		actingStep := 30;
		
	30: //finish command
		IF finished THEN
			IF actingFrame.SuccessFlag = 1 THEN
				actingStagingSlot := actingStagingSlot + 1;
			END_IF
			
			actingStep := 0; //stage next
		END_IF
		
END_CASE
END_METHOD

METHOD stagingSequence : BOOL
VAR_IN_OUT
	template : WoodBunkTable;
	magazine : MaterialStorage;
	table : WoodBunkTable;
	stagingSlot : INT;
	actingRobot : Robot;
	robotOutputs : ARRAY[1..50] OF INT;
	inspectionFrame : VisionFrame;
	actingStep : INT;
END_VAR
VAR_INPUT
	camera : INT;
END_VAR
VAR_OUTPUT
	fail : BOOL;
END_VAR
VAR
	finished : BOOL;
	slot : INT;
	templateArr : POINTER TO STRING;
END_VAR
VAR CONSTANT
	WIP : INT := 0;
	PASSED : INT := 1;
	FAILED : INT := 2;
END_VAR
IF table.isFull() OR stagingSlot > 10 THEN
	stagingSequence := TRUE;
	RETURN;
END_IF

templateArr := template.getSlotsAsArray();

//follow the template as is
IF NOT magazine.findSlot(materialID:= templateArr[stagingSlot], atSlot => slot) THEN
	fail := TRUE;
	RETURN;
END_IF

IF actingStep > 0 THEN
	finished := actingRobot.setCommandAndWait(A21.STAGE_BUNK, slot, stagingSlot, 0);
END_IF

CASE actingStep OF		
	0: //command
		IF actingRobot.inputs[5].10 THEN
			actingStep := 10;
		END_IF
		
	10: //request inspection
		tempInspectionSuite.frame.MaterialID := templateArr[stagingSlot];
		tempInspectionSuite.frame.CheckFor := 'ORIENTATION';
		tempInspectionSuite.frame.CameraNumber := camera;
	
		CreateJsonDocumentAuto(
			visionFrameData:= tempInspectionSuite.frame, 
			jsonDocument=> tempInspectionSuite.json);
		
		MEMCPY(
			ADR(tempInspectionSuite.data), 
			ADR(tempInspectionSuite.json), 
			MIN( SIZEOF(tempInspectionSuite.data), SIZEOF(tempInspectionSuite.json) ));
			
		TcpServer1Vision.queue(tempInspectionSuite.data);
		
		actingStep := 20;
	
	20: //fetch inspection data and parse
		actingRobot.setCommandAndWait(A21.STAGE_BUNK, slot, stagingSlot, 0);
		robotOutputs[4] := 0;
		
		IF NOT FrameIsValid(inspectionFrame) THEN
			RETURN;
		END_IF
		
		IF inspectionFrame.SuccessFlag = 1 THEN
			robotOutputs[4] := PASSED;
		ELSE
			robotOutputs[4] := FAILED;
		END_IF
		actingStep := 30;
		
	30: //finish command
		IF finished THEN
			IF inspectionFrame.SuccessFlag = 1 THEN
				stagingSlot := stagingSlot + 1;
			END_IF
			
			actingStep := 0;
		END_IF
END_CASE
END_METHOD

METHOD PROTECTED usesProcess : BOOL
VAR
	i : INT;
END_VAR
IF materialsArr = 0 THEN
	RETURN;
END_IF

FOR i:=0 TO GVL.maxPairs BY 1 DO
	IF PositionIsValid(materialsArr[i]) THEN
		usesProcess := TRUE;
		RETURN;
	END_IF
END_FOR
END_METHOD

END_FUNCTION_BLOCK

// ---- Sections/Concrete/AreaOutputEx.TcPOU
FUNCTION_BLOCK AreaOutputEx EXTENDS SectionEx
VAR_IN_OUT
	outputBuffer : ARRAY[*] OF Bundle;
END_VAR
VAR
	passConveyorPos (* AT %I* *) : REAL;
	failConveyorPos (* AT %I* *) : REAL;
	bufferConveyorPos (* AT %I* *) : REAL;
	
	step : (GET_RESULT, CHECK_RESULT, RESET);
	grade : (BYPASS, PASS, FAIL);
END_VAR
VAR
	gradeRequestString : STRING(1000);
	visionTimer : TON;
END_VAR
VAR_STAT CONSTANT
	visionTimeout : TIME := T#10S;
END_VAR

entryRefPos := bufferConveyorPos;
exitRefPos := MAX(passConveyorPos, failConveyorPos);

visionTimer(IN:= , PT:= visionTimeout, Q=> , ET=> );

SUPER^();

METHOD changeRobotsEOAT : BOOL
END_METHOD

METHOD gradeBundle : BOOL
VAR_INPUT
END_VAR
CASE grade OF
	PASS:
		//send to PASS output, LEFT
		
	BYPASS, FAIL:
		//send to FAIL output for manual correction, RIGHT
		
END_CASE
END_METHOD

METHOD initHardware : BOOL
conveyors := ADR(Hardware.allConveyors);
END_METHOD

METHOD PROTECTED load : BOOL
VAR_INPUT
	pair : REFERENCE TO PositionMaterials;
END_VAR
(*
loading takes place while the section is NOT active
materials are loaded for the next incoming bundle, not the current bundle - may differ for each section
*)
END_METHOD

METHOD PROTECTED process : BOOL
VAR
	gradingTcpData : TcpData;
END_VAR
VAR
	visionJson : STRING(1000);
	visionData : VisionFrame;
END_VAR
(*
area output process uses vision PC to determine if a bundle recipe was deployed correctly
1 output for passed bundles, 1 output for failed bundles, center is a buffer queue
*)

CASE step OF
	GET_RESULT:
		setConveyorMode(ConveyorMode.STOP); //stop at camera position (??)
		
		TcpServer1Vision.queue(gradingTcpData);
		step := CHECK_RESULT;
	
	CHECK_RESULT:
		setConveyorMode(ConveyorMode.STOP);
		visionTimer.IN := TRUE;
		
		TcpServer1Vision.fetch(gradingTcpData);
		
		IF NOT BufferIsEmpty(gradingTcpData.binaryData) THEN
			MEMCPY(ADR(visionJson), ADR(gradingTcpData.binaryData), MIN( SIZEOF(visionJson), SIZEOF(gradingTcpData.binaryData) ));
			VisionJsonParser(jsonString:= visionJson, visionData=> visionData);
		END_IF
		
		IF visionTimer.Q THEN
			visionTimer.IN := FALSE;
			grade := BYPASS;
		END_IF
	
	RESET:
		gradeBundle();
		process := TRUE;
		
END_CASE
END_METHOD

METHOD PROTECTED usesProcess : BOOL
VAR
	i : INT;
END_VAR
(*
IF materialsArr = 0 THEN
	RETURN;
END_IF

FOR i:=0 TO GVL.maxPairs BY 1 DO
	IF PositionIsValid(materialsArr[i]) THEN
		usesMaterial := TRUE;
		RETURN;		
	END_IF
END_FOR
*)
END_METHOD

END_FUNCTION_BLOCK
